PROGRAM TSM
VAR
	ResetHandler:FB_ResetSafetyHandler;
	ResetBtnOut AT %Q*:BOOL;
	AckDriveSafetyError AT %Q*:BOOL;
	EstopFromSafety AT %I*:BOOL;
	ErrorFromSafety AT %I*:BOOL;
	Override_Poti AT %I*:INT:=32700;
	DriveAckDelay:TOF;
	AllowEnable: BOOL;
	
	Door: FB_Door;
	DruckluftHS:FB_Actor;
	DruckluftSens:FB_Sensor;
	KMPumpe:FB_Actor;
	KSM_Spindel:FB_IFM_SV7200;
	KSM_Wanne:FB_Actor;
	Vakuum AT %Q*:bool;
	WanneFuellstand AT %I*:INT;
	
	BtnEStop:FB_BeckhoffTaster;
	BtnReset :FB_BeckhoffTaster;
	BtnGreen :FB_BeckhoffTaster;
	BtnRed :FB_BeckhoffTaster;
	Btn1 :FB_BeckhoffTaster; //Werkzeugwechsel
	Btn2 :FB_BeckhoffTaster;
	Btn3 :FB_BeckhoffTaster;
	Btn4 :FB_BeckhoffTaster;
	Btn5 :FB_BeckhoffTaster; //Open Door
	
	abyOutput: ARRAY [0..MAX_FAST_M_FUNC_OUTPUT_IDX] OF BYTE; 
END_VAR


//Aufrufe der Funktionen
IF BtnReset.wasRising() THEN
	ResetHandler.do_Reset();
	Door.Close();
END_IF

UPStart:=BtnGreen.isActive();
UPStop:=BtnRed.isActive();

ResetHandler(estop_ok_from_safety:=EstopFromSafety);
//IF NOT EstopFromSafety THEN PLCAxisEnable:=FALSE; END_IF

PlcFeedOverride:=INT_TO_UINT(Override_Poti/327);

Door();
MSG_WARNING_List[6]:=NOT Door.isLocked();
DruckluftHS();
DruckluftHS.setState(Druckluft_From_HMI);

//SpindelHSK(axisEnable:=PLCAxisEnable);

BtnEStop();
BtnReset();
BtnGreen();
BtnRed();
Btn1(schaltend:=TRUE);
Btn2(schaltend:=TRUE);
Btn3();
Btn4();
Btn5();

IF Btn5.wasRising() THEN
	PLCAxisEnable:=FALSE; 
	Door.Open();
END_IF


KSM_Spindel.setState(Btn1.isActive());
KSM_Wanne.setState(	NOT	Btn1.isActive()); //wur Wanne Spülen, wenn die Innenkühlung nicht aktiv ist
GlobalUniprec.strKSMt:=CONCAT(STR1:='KSM\n', STR2:=KSM_Spindel.getFlowString());
GlobalUniprec.strKSMt:=CONCAT(STR1:=GlobalUniprec.strKSMt ,STR2:='\n');
GlobalUniprec.strKSMt:=CONCAT(STR1:=GlobalUniprec.strKSMt , STR2:=KSM_Spindel.getTempString());
KSM_Spindel(Aktuator_Vorhanden:=TRUE);

Vakuum:=Btn2.isActive();

Mfct();

UPManualModebKeyNeg:=Btn3.isActive();
UPManualModebKeyPos:=Btn4.isActive();

METHOD doReset : BOOL
VAR_INPUT
END_VAR
END_METHOD

METHOD Mfct : BOOL
VAR_INPUT
END_VAR
VAR

	M :POINTER TO ARRAY [0..999] OF ST_TechnoAttributeData:=ADR(CNCSystem.Channel[0].M);
END_VAR
IF M^[7].bState_rw=TRUE THEN
	M^[7].bState_rw :=FALSE;
	Btn1.setON();
END_IF

IF M^[9].bState_rw=TRUE THEN
	M^[9].bState_rw :=FALSE;
	Btn1.setOFF();
END_IF
END_METHOD

END_PROGRAM

(* stored: Version 1.1.0.1, ProductVersion 3.1.4022.12
   POU TSM: Id {66d2a684-4b34-495f-b986-62233d7bcf49}, SpecialFunc None
   Method doReset: Id {16bea398-0baf-41a9-b487-5896b120f0fc}
   Method Mfct: Id {7d28f0d2-c8ff-4b68-a048-feb88c46d8b0} *)
